// TIA Portal project "Conveyor Speed Control Application with TIA Portal and SCADA" (V16)

(* hardware
DEVICE "PC-System_1"  SIMATIC PC station
   slot 0: "SIMATIC PC station"  Rail  SIMATIC PC-Station  V1.0
      slot 125: "Stationmanager"  Station_Manager  V6.0.4
   slot 1: "HMI_RT_1"  WinCC RT Professional  6AV2 105-0xxxx-xxxx  16.0.0.0
   slot 2: "IE general_1"  IE General  IE_CP  V8.2.0
DEVICE "S7-1200 station_1"  S7-1200 Station
   slot 0: "Rack_0"  S7-1200 Rack  Rack  V1.0
   slot 1: "PLC_1"  CPU 1212C DC/DC/DC  6ES7 212-1AE40-0XB0  V4.4
   slot 2: "AQ 2x14BIT_1"  6ES7 232-4HB30-0XB0  V1.0
   slot 3: "AQ 4x14BIT_1"  SM 1232 AQ4  6ES7 232-4HD30-0XB0  V1.0
DEVICE "HMI_1"  KTP700 Basic PN
   slot 0: "HMI_1"  KTP700 Basic PN  6AV2 123-2GB03-0AX0  16.0.0.0
   slot 1: "HMI_RT_2"  KTP700 Basic PN  6AV2 123-2GB03-0AX0  16.0.0.0
   slot 5: "HMI_1.IE_CP_1"  PROFINET Interface  16.0.0.0
      slot 1: "PROFINET Interface_1"  PROFINET Interface
         slot 1: "Port_1"  Port
*)

// ===== PLC "PLC_1"  CPU 1212C DC/DC/DC =====

VAR_GLOBAL   // PLC tag table "Default tag table"
   "Startup_mem" AT %M10.0 : Bool;
END_VAR

VAR_GLOBAL   // PLC tag table "ANALLOG"
   "BAND2" AT %QW96 : Word;
   "BAND3" AT %QW98 : Int;
   "SİSTEM ÇAŞMA DURUMU" AT %QW30 : Int;
END_VAR

VAR_GLOBAL   // PLC tag table "İnputs"
   "Start_But" AT %I0.0 : Bool;
   "Stop_But" AT %I0.1 : Bool;
   "Start_But_Analog" AT %I0.2 : Bool;
   "Stop_But_Analog" AT %I0.3 : Bool;
   "Start_laması" AT %I0.4 : Bool;
   "Stop_lambası" AT %I0.5 : Bool;
END_VAR

VAR_GLOBAL   // PLC tag table "Outputs"
   "Lamba" AT %Q0.0 : Bool;
   "Band_konveyör" AT %Q0.2 : Bool;
   "Band_konveyör_1" AT %Q0.3 : Bool;
   "Lamba_1" AT %Q0.4 : Bool;
   "konveyör_1" AT %Q0.5 : Bool;
   "konveyör_2" AT %Q0.6 : Bool;
   "konveyör_3" AT %Q0.7 : Bool;
   "konveyör_4" AT %Q1.0 : Bool;
END_VAR

DATA_BLOCK "Datalar"   // DB1
{ S7_Optimized_Access := 'TRUE' }
VERSION : 0.1
   VAR
      Hmi_Start_BUt : Bool;
      Hmi_Stop_BUt : Bool;
      Hmi_jogg_BUt : Bool;
      Band_konveyör : Bool;
      yardımcı_Mem_1 : Bool;
      yardımcı_Mem_2 : Bool;
      Hmi_Toggle_button : Bool;
      Hmi_Azalt_button : Bool;
      Hmi_Artır_button : Bool;
      Hız_değeri : Int;
      band_konveyör_2 : Bool;
      lamba : Bool;
      TEMP_1 : Bool;
      TEMP_2 : Bool;
      TEMP_3 : Bool;
      TEMP_4 : Bool;
      TEMP_5 : Bool;
      KONVEYÖR_HATTI : Struct
         Hmi_Start : Bool;
         Hmi_Stop : Bool;
         Hmi_Merker1 : Bool;
         Sayma_Değeri : Int;
         Hmi_Start_Analog : Bool;
         Hmi_Stop_Analog : Bool;
         Start_Stop_button : Bool;
         Start_Stop_Mem : Bool;
         "Sistem_durum bilgisi" : Int;
      END_STRUCT;
   END_VAR
BEGIN
END_DATA_BLOCK

// folder: System blocks/Program resources

DATA_BLOCK "time_1"   // DB2
{ S7_Optimized_Access := 'TRUE' }
AUTHOR : Simatic
FAMILY : IEC
NAME : IEC_TMR
VERSION : 1.0
// stored: InstanceOfName IEC_TIMER
"IEC_TIMER"
BEGIN
END_DATA_BLOCK

DATA_BLOCK "time_2"   // DB3
{ S7_Optimized_Access := 'TRUE' }
AUTHOR : Simatic
FAMILY : IEC
NAME : IEC_TMR
VERSION : 1.0
// stored: InstanceOfName IEC_TIMER
"IEC_TIMER"
BEGIN
END_DATA_BLOCK

// folder: (top level)

FUNCTION "üretim Hattı 2" : Void   // FC1, LAD
{ S7_Optimized_Access := 'TRUE' }
VERSION : 0.1
BEGIN

REGION Network 1
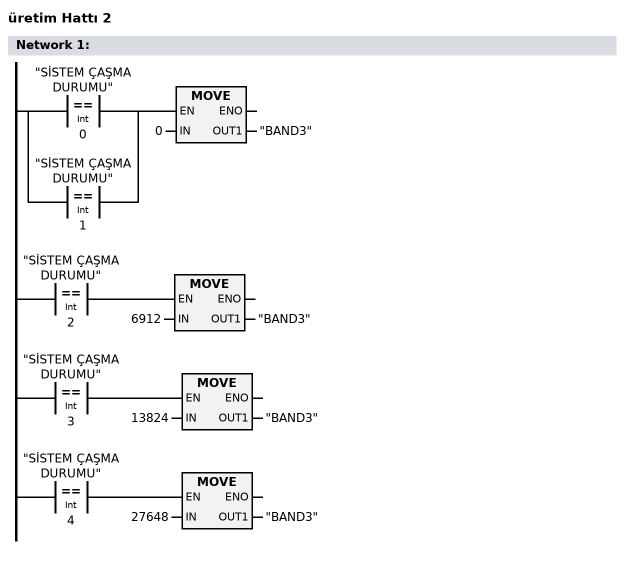
   RUNG wire#powerrail
      { S7_Templates := "SrcType := Int" } EQ_Contact(in1 := "SİSTEM ÇAŞMA DURUMU", in2 := 0)
      wire#w1
      Move(in := 0, out1 => "BAND3")
   END_RUNG
   RUNG wire#powerrail
      { S7_Templates := "SrcType := Int" } EQ_Contact(in1 := "SİSTEM ÇAŞMA DURUMU", in2 := 1)
   END_RUNG wire#w1
   RUNG wire#powerrail
      { S7_Templates := "SrcType := Int" } EQ_Contact(in1 := "SİSTEM ÇAŞMA DURUMU", in2 := 2)
      Move(in := 6912, out1 => "BAND3")
   END_RUNG
   RUNG wire#powerrail
      { S7_Templates := "SrcType := Int" } EQ_Contact(in1 := "SİSTEM ÇAŞMA DURUMU", in2 := 3)
      Move(in := 13824, out1 => "BAND3")
   END_RUNG
   RUNG wire#powerrail
      { S7_Templates := "SrcType := Int" } EQ_Contact(in1 := "SİSTEM ÇAŞMA DURUMU", in2 := 4)
      Move(in := 27648, out1 => "BAND3")
   END_RUNG
   // the same network as SCL:
   IF ("SİSTEM ÇAŞMA DURUMU" = 0) OR ("SİSTEM ÇAŞMA DURUMU" = 1) THEN "BAND3" := 0; END_IF;
   IF "SİSTEM ÇAŞMA DURUMU" = 2 THEN "BAND3" := 6912; END_IF;
   IF "SİSTEM ÇAŞMA DURUMU" = 3 THEN "BAND3" := 13824; END_IF;
   IF "SİSTEM ÇAŞMA DURUMU" = 4 THEN "BAND3" := 27648; END_IF;
END_REGION
END_FUNCTION

FUNCTION "Üretin_hattı_3" : Void   // FC2, LAD
{ S7_Optimized_Access := 'TRUE' }
VERSION : 0.1
BEGIN

REGION Network 1: Sistem Start Stop
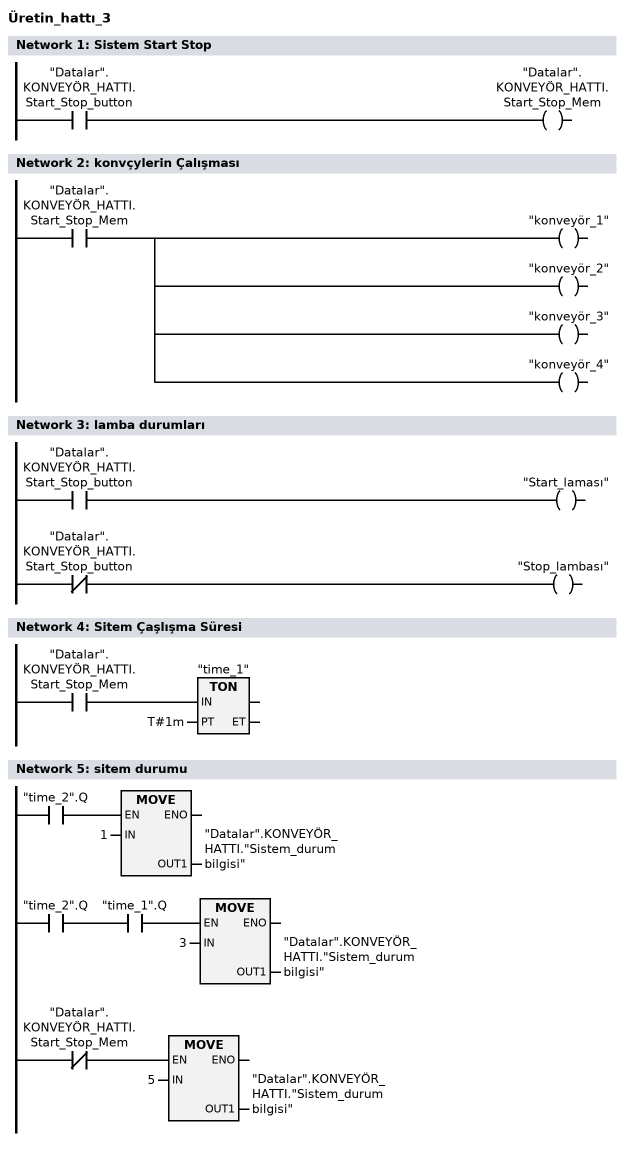
   RUNG wire#powerrail
      Contact( "Datalar".KONVEYÖR_HATTI.Start_Stop_button )
      Coil( "Datalar".KONVEYÖR_HATTI.Start_Stop_Mem )
   END_RUNG
   // the same network as SCL:
   "Datalar".KONVEYÖR_HATTI.Start_Stop_Mem := "Datalar".KONVEYÖR_HATTI.Start_Stop_button;
END_REGION

REGION Network 2: konvçylerin Çalışması
   RUNG wire#powerrail
      Contact( "Datalar".KONVEYÖR_HATTI.Start_Stop_Mem )
      wire#w1
      Coil( "konveyör_1" )
   END_RUNG
   RUNG wire#w1
      Coil( "konveyör_2" )
   END_RUNG
   RUNG wire#w1
      Coil( "konveyör_3" )
   END_RUNG
   RUNG wire#w1
      Coil( "konveyör_4" )
   END_RUNG
   // the same network as SCL:
   "konveyör_1" := "Datalar".KONVEYÖR_HATTI.Start_Stop_Mem;
   "konveyör_2" := "Datalar".KONVEYÖR_HATTI.Start_Stop_Mem;
   "konveyör_3" := "Datalar".KONVEYÖR_HATTI.Start_Stop_Mem;
   "konveyör_4" := "Datalar".KONVEYÖR_HATTI.Start_Stop_Mem;
END_REGION

REGION Network 3: lamba durumları
   RUNG wire#powerrail
      Contact( "Datalar".KONVEYÖR_HATTI.Start_Stop_button )
      Coil( "Start_laması" )
   END_RUNG
   RUNG wire#powerrail
      I_Contact( "Datalar".KONVEYÖR_HATTI.Start_Stop_button )
      Coil( "Stop_lambası" )
   END_RUNG
   // the same network as SCL:
   "Start_laması" := "Datalar".KONVEYÖR_HATTI.Start_Stop_button;
   "Stop_lambası" := NOT "Datalar".KONVEYÖR_HATTI.Start_Stop_button;
END_REGION

REGION Network 4: Sitem Çaşlışma Süresi
   "time_1".TON(IN := "Datalar".KONVEYÖR_HATTI.Start_Stop_Mem, PT := T#1m);
END_REGION

REGION Network 5: sitem durumu
   RUNG wire#powerrail
      Contact( "time_2".Q )
      Move(in := 1, out1 => "Datalar".KONVEYÖR_HATTI."Sistem_durum bilgisi")
   END_RUNG
   RUNG wire#powerrail
      Contact( "time_2".Q )
      Contact( "time_1".Q )
      Move(in := 3, out1 => "Datalar".KONVEYÖR_HATTI."Sistem_durum bilgisi")
   END_RUNG
   RUNG wire#powerrail
      I_Contact( "Datalar".KONVEYÖR_HATTI.Start_Stop_Mem )
      Move(in := 5, out1 => "Datalar".KONVEYÖR_HATTI."Sistem_durum bilgisi")
   END_RUNG
   // the same network as SCL:
   IF "time_2".Q THEN "Datalar".KONVEYÖR_HATTI."Sistem_durum bilgisi" := 1; END_IF;
   IF "time_2".Q AND "time_1".Q THEN "Datalar".KONVEYÖR_HATTI."Sistem_durum bilgisi" := 3; END_IF;
   IF NOT "Datalar".KONVEYÖR_HATTI.Start_Stop_Mem THEN
       "Datalar".KONVEYÖR_HATTI."Sistem_durum bilgisi" := 5;
   END_IF;
END_REGION
END_FUNCTION

ORGANIZATION_BLOCK "Main"   // OB1, LAD, ProgramCycle
TITLE = "Main Program Sweep (Cycle)"
{ S7_Optimized_Access := 'TRUE' }
VERSION : 0.1
   VAR_INPUT
      Initial_Call : Bool;   // Initial call of this OB
      Remanence : Bool;   // =True, if remanent data are available
   END_VAR
   VAR_TEMP   // added for the SCL form of the ladder/FBD networks
      _w1 : Bool;
      _w2 : Bool;
   END_VAR
BEGIN

REGION Network 1: ÜRETİM HATTI 2
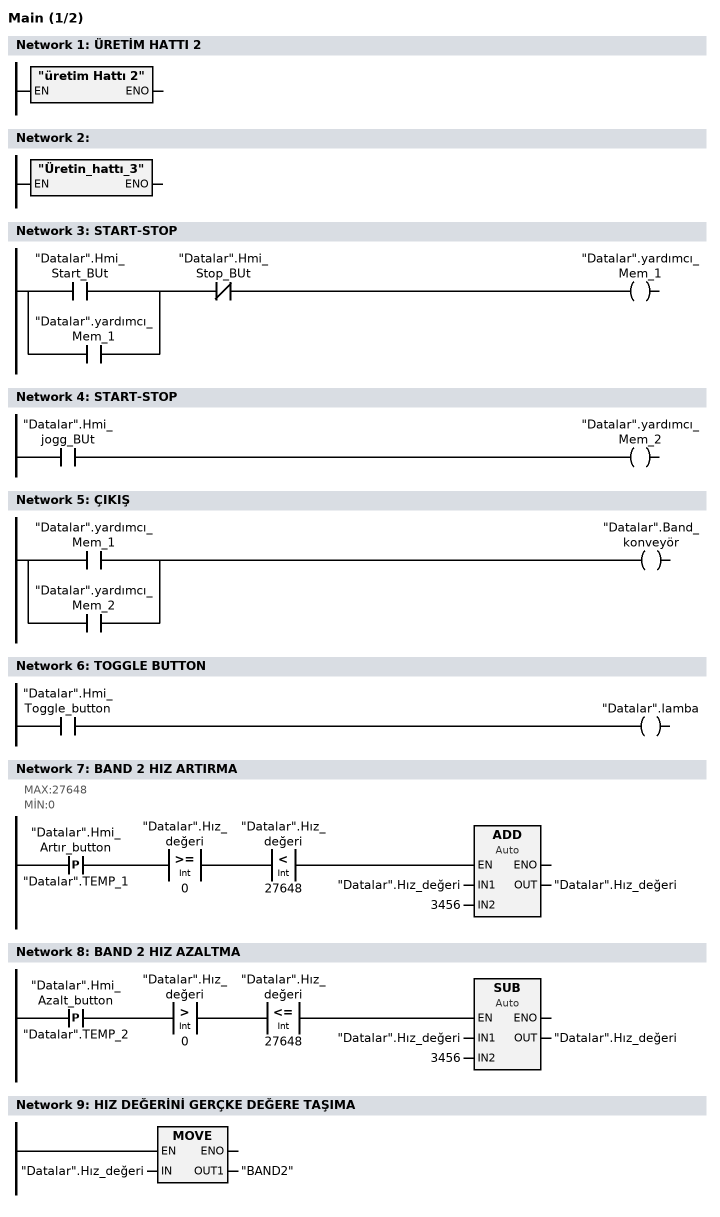
   RUNG wire#powerrail
      "üretim Hattı 2"()
   END_RUNG
   // the same network as SCL:
   "üretim Hattı 2"();
END_REGION

REGION Network 2
   RUNG wire#powerrail
      "Üretin_hattı_3"()
   END_RUNG
   // the same network as SCL:
   "Üretin_hattı_3"();
END_REGION

REGION Network 3: START-STOP
   RUNG wire#powerrail
      Contact( "Datalar".Hmi_Start_BUt )
      wire#w1
      I_Contact( "Datalar".Hmi_Stop_BUt )
      Coil( "Datalar".yardımcı_Mem_1 )
   END_RUNG
   RUNG wire#powerrail
      Contact( "Datalar".yardımcı_Mem_1 )
   END_RUNG wire#w1
   // the same network as SCL:
   "Datalar".yardımcı_Mem_1 := ("Datalar".Hmi_Start_BUt OR "Datalar".yardımcı_Mem_1) AND NOT "Datalar".Hmi_Stop_BUt;
END_REGION

REGION Network 4: START-STOP
   RUNG wire#powerrail
      Contact( "Datalar".Hmi_jogg_BUt )
      Coil( "Datalar".yardımcı_Mem_2 )
   END_RUNG
   // the same network as SCL:
   "Datalar".yardımcı_Mem_2 := "Datalar".Hmi_jogg_BUt;
END_REGION

REGION Network 5: ÇIKIŞ
   RUNG wire#powerrail
      Contact( "Datalar".yardımcı_Mem_1 )
      wire#w1
      Coil( "Datalar".Band_konveyör )
   END_RUNG
   RUNG wire#powerrail
      Contact( "Datalar".yardımcı_Mem_2 )
   END_RUNG wire#w1
   // the same network as SCL:
   "Datalar".Band_konveyör := "Datalar".yardımcı_Mem_1 OR "Datalar".yardımcı_Mem_2;
END_REGION

REGION Network 6: TOGGLE BUTTON
   RUNG wire#powerrail
      Contact( "Datalar".Hmi_Toggle_button )
      Coil( "Datalar".lamba )
   END_RUNG
   // the same network as SCL:
   "Datalar".lamba := "Datalar".Hmi_Toggle_button;
END_REGION

REGION Network 7: BAND 2 HIZ ARTIRMA
   // MAX:27648
   // MİN:0
   RUNG wire#powerrail
      P_Contact(operand := "Datalar".Hmi_Artır_button, bit := "Datalar".TEMP_1)
      { S7_Templates := "SrcType := Int" } GE_Contact(in1 := "Datalar".Hız_değeri, in2 := 0)
      { S7_Templates := "SrcType := Int" } LT_Contact(in1 := "Datalar".Hız_değeri, in2 := 27648)
      Add(in1 := "Datalar".Hız_değeri, in2 := 3456, out => "Datalar".Hız_değeri)
   END_RUNG
   // the same network as SCL:
   #_w1 := "Datalar".Hmi_Artır_button AND NOT "Datalar".TEMP_1;   // rising edge of "Datalar".Hmi_Artır_button
   "Datalar".TEMP_1 := "Datalar".Hmi_Artır_button;
   IF #_w1 AND ("Datalar".Hız_değeri >= 0) AND ("Datalar".Hız_değeri < 27648) THEN
       "Datalar".Hız_değeri := "Datalar".Hız_değeri + 3456;
   END_IF;
END_REGION

REGION Network 8: BAND 2 HIZ AZALTMA
   RUNG wire#powerrail
      P_Contact(operand := "Datalar".Hmi_Azalt_button, bit := "Datalar".TEMP_2)
      { S7_Templates := "SrcType := Int" } GT_Contact(in1 := "Datalar".Hız_değeri, in2 := 0)
      { S7_Templates := "SrcType := Int" } LE_Contact(in1 := "Datalar".Hız_değeri, in2 := 27648)
      Sub(in1 := "Datalar".Hız_değeri, in2 := 3456, out => "Datalar".Hız_değeri)
   END_RUNG
   // the same network as SCL:
   #_w1 := "Datalar".Hmi_Azalt_button AND NOT "Datalar".TEMP_2;   // rising edge of "Datalar".Hmi_Azalt_button
   "Datalar".TEMP_2 := "Datalar".Hmi_Azalt_button;
   IF #_w1 AND ("Datalar".Hız_değeri > 0) AND ("Datalar".Hız_değeri <= 27648) THEN
       "Datalar".Hız_değeri := "Datalar".Hız_değeri - 3456;
   END_IF;
END_REGION

REGION Network 9: HIZ DEĞERİNİ GERÇKE DEĞERE TAŞIMA
   RUNG wire#powerrail
      Move(in := "Datalar".Hız_değeri, out1 => "BAND2")
   END_RUNG
   // the same network as SCL:
   "BAND2" := "Datalar".Hız_değeri;
END_REGION

REGION Network 10: KONYEYÖR HATTINI ÇALIŞTIRMA 1
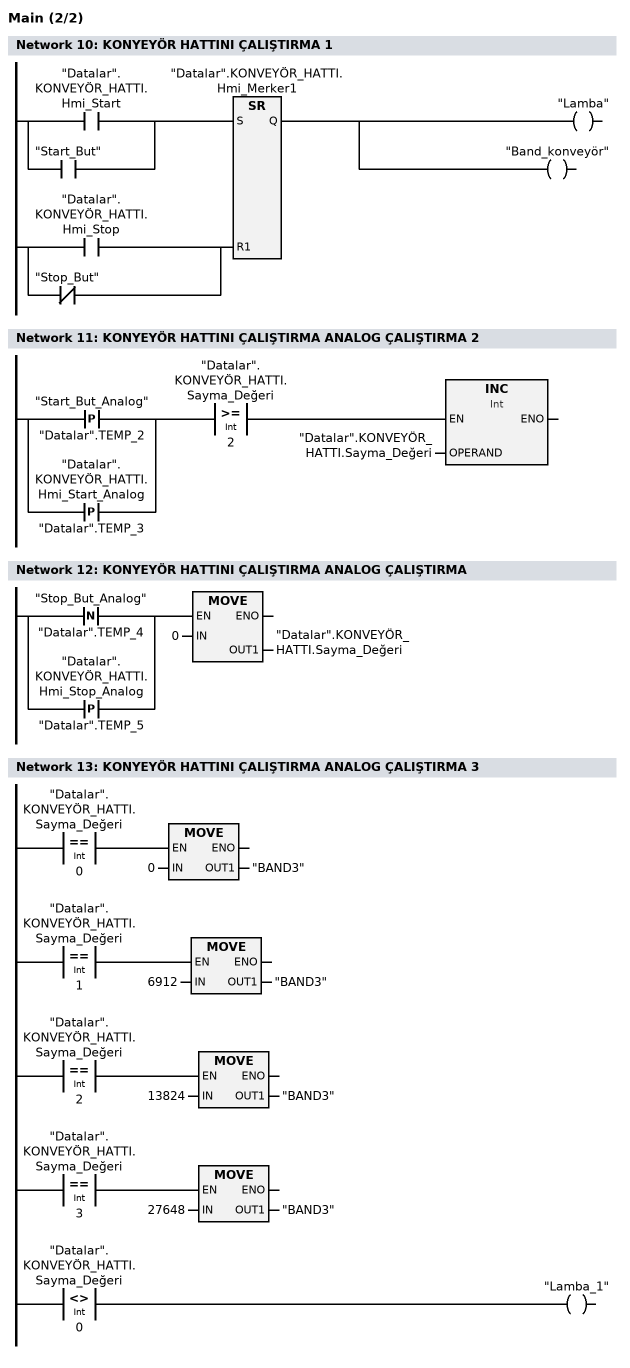
   RUNG wire#powerrail
      Contact( "Datalar".KONVEYÖR_HATTI.Hmi_Start )
      wire#w1
      S_SR(operand := "Datalar".KONVEYÖR_HATTI.Hmi_Merker1, r1 := wire#w2)
      wire#w3
      Coil( "Lamba" )
   END_RUNG
   RUNG wire#powerrail
      Contact( "Start_But" )
   END_RUNG wire#w1
   RUNG wire#powerrail
      Contact( "Datalar".KONVEYÖR_HATTI.Hmi_Stop )
   END_RUNG wire#w2
   RUNG wire#powerrail
      I_Contact( "Stop_But" )
   END_RUNG wire#w2
   RUNG wire#w3
      Coil( "Band_konveyör" )
   END_RUNG
   // the same network as SCL:
   IF "Datalar".KONVEYÖR_HATTI.Hmi_Start OR "Start_But" THEN
       "Datalar".KONVEYÖR_HATTI.Hmi_Merker1 := TRUE;   // SR flip-flop
   END_IF;
   IF "Datalar".KONVEYÖR_HATTI.Hmi_Stop OR NOT "Stop_But" THEN
       "Datalar".KONVEYÖR_HATTI.Hmi_Merker1 := FALSE;
   END_IF;
   "Lamba" := "Datalar".KONVEYÖR_HATTI.Hmi_Merker1;
   "Band_konveyör" := "Datalar".KONVEYÖR_HATTI.Hmi_Merker1;
END_REGION

REGION Network 11: KONYEYÖR HATTINI ÇALIŞTIRMA ANALOG ÇALIŞTIRMA 2
   RUNG wire#powerrail
      P_Contact(operand := "Start_But_Analog", bit := "Datalar".TEMP_2)
      wire#w1
      { S7_Templates := "SrcType := Int" } GE_Contact(in1 := "Datalar".KONVEYÖR_HATTI.Sayma_Değeri, in2 := 2)
      { S7_Templates := "DestType := Int" } Inc( "Datalar".KONVEYÖR_HATTI.Sayma_Değeri )
   END_RUNG
   RUNG wire#powerrail
      P_Contact(operand := "Datalar".KONVEYÖR_HATTI.Hmi_Start_Analog, bit := "Datalar".TEMP_3)
   END_RUNG wire#w1
   // the same network as SCL:
   #_w1 := "Start_But_Analog" AND NOT "Datalar".TEMP_2;   // rising edge of "Start_But_Analog"
   "Datalar".TEMP_2 := "Start_But_Analog";
   #_w2 := "Datalar".KONVEYÖR_HATTI.Hmi_Start_Analog AND NOT "Datalar".TEMP_3;   // rising edge of "Datalar".KONVEYÖR_HATTI.Hmi_Start_Analog
   "Datalar".TEMP_3 := "Datalar".KONVEYÖR_HATTI.Hmi_Start_Analog;
   IF (#_w1 OR #_w2) AND ("Datalar".KONVEYÖR_HATTI.Sayma_Değeri >= 2) THEN
       "Datalar".KONVEYÖR_HATTI.Sayma_Değeri := "Datalar".KONVEYÖR_HATTI.Sayma_Değeri + 1;
   END_IF;
END_REGION

REGION Network 12: KONYEYÖR HATTINI ÇALIŞTIRMA ANALOG ÇALIŞTIRMA
   RUNG wire#powerrail
      N_Contact(operand := "Stop_But_Analog", bit := "Datalar".TEMP_4)
      wire#w1
      Move(in := 0, out1 => "Datalar".KONVEYÖR_HATTI.Sayma_Değeri)
   END_RUNG
   RUNG wire#powerrail
      P_Contact(operand := "Datalar".KONVEYÖR_HATTI.Hmi_Stop_Analog, bit := "Datalar".TEMP_5)
   END_RUNG wire#w1
   // the same network as SCL:
   #_w1 := NOT "Stop_But_Analog" AND "Datalar".TEMP_4;   // falling edge of "Stop_But_Analog"
   "Datalar".TEMP_4 := "Stop_But_Analog";
   #_w2 := "Datalar".KONVEYÖR_HATTI.Hmi_Stop_Analog AND NOT "Datalar".TEMP_5;   // rising edge of "Datalar".KONVEYÖR_HATTI.Hmi_Stop_Analog
   "Datalar".TEMP_5 := "Datalar".KONVEYÖR_HATTI.Hmi_Stop_Analog;
   IF #_w1 OR #_w2 THEN "Datalar".KONVEYÖR_HATTI.Sayma_Değeri := 0; END_IF;
END_REGION

REGION Network 13: KONYEYÖR HATTINI ÇALIŞTIRMA ANALOG ÇALIŞTIRMA 3
   RUNG wire#powerrail
      { S7_Templates := "SrcType := Int" } EQ_Contact(in1 := "Datalar".KONVEYÖR_HATTI.Sayma_Değeri, in2 := 0)
      Move(in := 0, out1 => "BAND3")
   END_RUNG
   RUNG wire#powerrail
      { S7_Templates := "SrcType := Int" } EQ_Contact(in1 := "Datalar".KONVEYÖR_HATTI.Sayma_Değeri, in2 := 1)
      Move(in := 6912, out1 => "BAND3")
   END_RUNG
   RUNG wire#powerrail
      { S7_Templates := "SrcType := Int" } EQ_Contact(in1 := "Datalar".KONVEYÖR_HATTI.Sayma_Değeri, in2 := 2)
      Move(in := 13824, out1 => "BAND3")
   END_RUNG
   RUNG wire#powerrail
      { S7_Templates := "SrcType := Int" } EQ_Contact(in1 := "Datalar".KONVEYÖR_HATTI.Sayma_Değeri, in2 := 3)
      Move(in := 27648, out1 => "BAND3")
   END_RUNG
   RUNG wire#powerrail
      { S7_Templates := "SrcType := Int" } NE_Contact(in1 := "Datalar".KONVEYÖR_HATTI.Sayma_Değeri, in2 := 0)
      Coil( "Lamba_1" )
   END_RUNG
   // the same network as SCL:
   IF "Datalar".KONVEYÖR_HATTI.Sayma_Değeri = 0 THEN "BAND3" := 0; END_IF;
   IF "Datalar".KONVEYÖR_HATTI.Sayma_Değeri = 1 THEN "BAND3" := 6912; END_IF;
   IF "Datalar".KONVEYÖR_HATTI.Sayma_Değeri = 2 THEN "BAND3" := 13824; END_IF;
   IF "Datalar".KONVEYÖR_HATTI.Sayma_Değeri = 3 THEN "BAND3" := 27648; END_IF;
   "Lamba_1" := "Datalar".KONVEYÖR_HATTI.Sayma_Değeri <> 0;
END_REGION
END_ORGANIZATION_BLOCK

ORGANIZATION_BLOCK "Startup"   // OB100, LAD, Startup
TITLE = "Complete Restart"
{ S7_Optimized_Access := 'TRUE' }
VERSION : 0.1
   VAR_INPUT
      LostRetentive : Bool;   // True if retentive data are lost
      LostRTC : Bool;   // True if date and time are lost
   END_VAR
BEGIN

REGION Network 1
   // plc Stop modula alıp terkara run veririsek 25saniye sonra run oluca
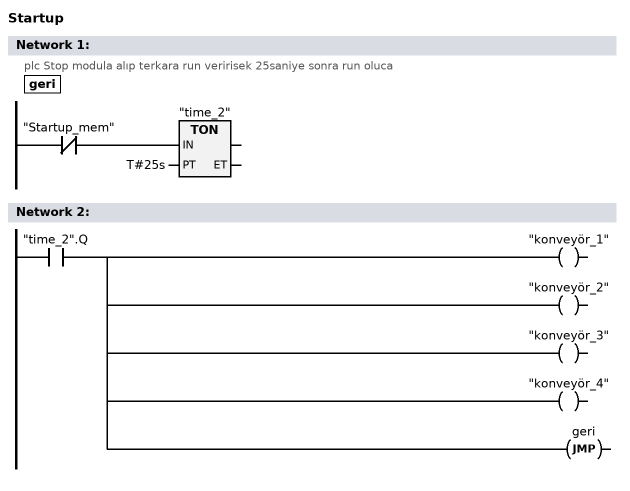
   geri:
   "time_2".TON(IN := NOT "Startup_mem", PT := T#25s);
END_REGION

REGION Network 2
   RUNG wire#powerrail
      Contact( "time_2".Q )
      wire#w1
      Coil( "konveyör_1" )
   END_RUNG
   RUNG wire#w1
      Coil( "konveyör_2" )
   END_RUNG
   RUNG wire#w1
      Coil( "konveyör_3" )
   END_RUNG
   RUNG wire#w1
      Coil( "konveyör_4" )
   END_RUNG
   RUNG wire#w1
      JumpCoil( geri )
   END_RUNG
   // the same network as SCL:
   "konveyör_1" := "time_2".Q;
   "konveyör_2" := "time_2".Q;
   "konveyör_3" := "time_2".Q;
   "konveyör_4" := "time_2".Q;
   IF "time_2".Q THEN GOTO geri; END_IF;
END_REGION
END_ORGANIZATION_BLOCK

(* ===== HMI "HMI_RT_1" =====
system functions are stored by id; their names below are inferred from use
connection "HMI_Connection_1": S71200_TCP_IP, SCADA_S7_1200

HMI tags "Default tag table"
   "a" : Bool = PLC a AT %I0.0, 500 ms
   "Datalar_Hmi_Start_BUt" : Bool = PLC Datalar.Hmi_Start_BUt, 500 ms
   "Datalar_Hmi_Stop_BUt" : Bool = PLC Datalar.Hmi_Stop_BUt, 500 ms
   "Datalar_Hmi_jogg_BUt" : Bool = PLC Datalar.Hmi_jogg_BUt, 500 ms
   "Datalar_Hmi_Toggle_button" : Bool = PLC Datalar.Hmi_Toggle_button, 500 ms
   "Datalar_Hmi_Artır_button" : Bool = PLC Datalar.Hmi_Artır_button, 500 ms
   "Datalar_Hmi_Azalt_button" : Bool = PLC Datalar.Hmi_Azalt_button, 500 ms
   "Datalar_KONVEYÖR_HATTI_Hmi_Start" : Bool = PLC Datalar.KONVEYÖR_HATTI.Hmi_Start, 500 ms
   "Datalar_KONVEYÖR_HATTI_Hmi_Stop" : Bool = PLC Datalar.KONVEYÖR_HATTI.Hmi_Stop, 500 ms
   "Lamba" : Bool = PLC Lamba AT %Q0.0, 500 ms
   "Band_konveyör" : Bool = PLC Band_konveyör AT %Q0.2, 500 ms
   "BAND3" : Int = PLC BAND3 AT %QW98, 500 ms
   "SİSTEMÇAŞMADURUMU" : Int = PLC "SİSTEM ÇAŞMA DURUMU" AT %QW30, 500 ms
   "Datalar_KONVEYÖR_HATTI_Sistem_durumbilgisi" : Int = PLC Datalar.KONVEYÖR_HATTI."Sistem_durum bilgisi", 500 ms
   "Datalar_KONVEYÖR_HATTI_Start_Stop_button" : Bool = PLC Datalar.KONVEYÖR_HATTI.Start_Stop_button, 500 ms

screen "Ana Sayfa" 1024x768
   Button "Button_1" at 118,107 size 107x63; TextOff 'START BUT'
   Button "Button_2" at 250,109 size 107x63; TextOff 'STOP BUT'
      on PressLeft: SetBit("Datalar_Hmi_Stop_BUt")
      on ReleaseLeft: ResetBit("Datalar_Hmi_Stop_BUt")
   Button "Button_3" at 390,109 size 107x63; TextOff 'JOGG BUT'
      on PressLeft: SetBit("Datalar_Hmi_jogg_BUt")
      on ReleaseLeft: ResetBit("Datalar_Hmi_jogg_BUt")
   RoundButton "Round button_1" at 299,306 size 93x93; Text 'TOGGLE BUTTON'
      on Click: InvertBit("Datalar_Hmi_Toggle_button")
   TextField "Text field_1" at 262,17 size 144x23; Text 'BUTTON TİPLERİ'
   Button "Button_4" at 156,282 size 76x60; TextOff 'Text'; PictureOff "Up_Arrow"
      on PressLeft: SetBit("Datalar_Hmi_Artır_button")
      on ReleaseLeft: ResetBit("Datalar_Hmi_Artır_button")
   Button "Button_5" at 162,399 size 72x66; TextOff 'Text'; PictureOff "Down_Arrow"
      on PressLeft: SetBit("Datalar_Hmi_Azalt_button")
      on ReleaseLeft: ResetBit("Datalar_Hmi_Azalt_button")
   TextField "Text field_2" at 159,246 size 80x21; Text 'HIZ ARTIR'
   TextField "Text field_3" at 159,369 size 82x21; Text 'HIZ AZALT'

screen "Üretim Hattı" 1024x768
   GraphicView "Graphic view_1" at 155,46 size 299x183; Picture "Graphic_1"
   TextField "Text field_1" at 259,15 size 102x19; Text 'Üretim Hattı'
   Button "Button_1" at 512,70 size 99x52; TextOff 'Start'
      on PressLeft: SetBit("Datalar_KONVEYÖR_HATTI_Hmi_Start")
      on ReleaseLeft: ResetBit("Datalar_KONVEYÖR_HATTI_Hmi_Start")
   Button "Button_2" at 686,70 size 99x52; TextOff 'Stop'
      on PressLeft: SetBit("Datalar_KONVEYÖR_HATTI_Hmi_Stop")
      on ReleaseLeft: ResetBit("Datalar_KONVEYÖR_HATTI_Hmi_Stop")
   GraphicView "Graphic view_2" at 258,112 size 97x127; Picture "Graphic_2"
   Circle "Circle_1" at 268,132 size 25x25
      Visibility <- "Lamba"
      Appearance <- "BAND3"
   Circle "Circle_2" at 310,132 size 24x24
      Appearance <- "BAND3"
   TextField "Text field_2" at 259,241 size 110x19; Text 'sistem Çalışıyor'
      Visibility <- "Band_konveyör"
   TextField "Text field_3" at 259,271 size 108x19; Text 'sistem Duruyor'
      Visibility <- "Band_konveyör"
   ListBox "List box_1" at 422,171 size 300x15; Text0 'Text1'
      SelectedIndex <- "BAND3"
      PropertyAnimation0 <- "BAND3"

screen "Üreti Hattı_2" 1024x768
   GraphicView "Graphic view_1" at 155,46 size 299x183; Picture "Graphic_1"
   TextField "Text field_1" at 259,15 size 102x19; Text 'Üretim Hattı'
   GraphicView "Graphic view_2" at 258,112 size 97x127; Picture "Graphic_2"
   Circle "Circle_1" at 268,132 size 25x25
      Visibility <- "Lamba"
      Appearance <- "BAND3"
   Circle "Circle_2" at 310,132 size 24x24
      Appearance <- "BAND3"
   ListBox "List box_1" at 109,241 size 461x68; Text0 'SİSTEM DURUYOR'; Text1 'SİSTEM YAVAŞ HIZDA ÇALIŞIYOR'; Text2 'SİSTEM ORTA HIZDA ÇALIŞIYOR'; Text3 'SİSTEM YÜKSEK HIZDA ÇALIŞIYOR'
      SelectedIndex <- "SİSTEMÇAŞMADURUMU"
   Button "Button_1" at 509,60 size 124x65; TextOff 'Start'
   Button "Button_2" at 672,57 size 124x65; TextOff 'Stop'
   ComboBox "Combo box_1" at 120,339 size 439x30; Text0 'SİSTEM DURUYOR'; Text1 'SİSTEM YAVAŞ HIZDA ÇALIŞIYOR'; Text2 'SİSTEM ORTA HIZDA ÇALIŞIYOR'; Text3 'SİSTEM YÜKSEK HIZDA ÇALIŞIYOR'
      SelectedIndex <- "SİSTEMÇAŞMADURUMU"

screen "Üretim hattı_3" 1024x768
   RoundButton "Round button_1" at 42,117 size 83x83; Text 'Start Stop'
      on Click: InvertBit("Datalar_KONVEYÖR_HATTI_Start_Stop_button")
   GraphicView "Graphic view_1" at 200,35 size 299x183; Picture "Graphic_1"
   GraphicView "Graphic view_2" at 303,101 size 97x127; Picture "Graphic_2"
   CheckBox "Check box_1" at 94,266 size 236x93; Text0 'Sistem ilk konuma Alındı'; Text1 'Sistem Bir dk dan fazla çalıştı'; Text2 'Sistem Durdu'
      ProcessValue <- "Datalar_KONVEYÖR_HATTI_Sistem_durumbilgisi"
   TextField "Text field_1" at 111,243 size 90x19; Text 'Onay Kutusu'
*)

(* ===== HMI "HMI_RT_2" =====
system functions are stored by id; their names below are inferred from use
connection "HMI_Connection_2": ETHERNET, SMART_S7_1200_OMS

HMI tags "Default tag table"
   "Tag_ScreenNumber" : UInt, internal

Template "Template_1" 800x480
   Button "Exit" at 714,429 size 71x50; TextOff 'Exit'; PictureOff "ExitRuntime_KTP700_Basic_PN_TR"; PictureOn "ExitRuntime_KTP700_Basic_PN_TR"
      on Release: StopRuntime(0)
   Button "Template_Button" at 614,429 size 71x50; TextOff 'Text'
   Button "Template_Button_1" at 514,429 size 71x50; TextOff 'Text'
   Button "Template_Button_2" at 414,429 size 71x50; TextOff 'Text'
   Button "Template_Button_3" at 314,429 size 71x50; TextOff 'Text'
   Button "Template_Button_4" at 214,429 size 71x50; TextOff 'Text'
   Button "Template_Button_5" at 114,429 size 71x50; TextOff 'Text'
   Button "Start screen" at 14,429 size 71x50; TextOff 'Start screen'; PictureOff "NavigateHome_KTP700_Basic_PN_TR"; PictureOn "NavigateHome_KTP700_Basic_PN_TR"
      on Release: ActivateScreen("Root screen", 0)
   SymbolicIOField "Symbolic_IO_Field_Screen" at 93,9 size 600x33; TextOff '0'; TextOn '1'; TextList "TextList_ScreenNames"
      ProcessValue <- "Tag_ScreenNumber"
      on Change: ActivateScreenByNumber("Tag_ScreenNumber", 0)
   DateTimeField "HmiScreenItemData" at 695,25 size 105x25
   DateTimeField "HmiScreenItemData_1" at 695,0 size 105x25
   GraphicView "Logo" at 0,0 size 91x51; Picture "Logo of HMI_1"

screen "Root screen" 800x480, template "Template_1"
   on GenerateScreen: SetTag("Tag_ScreenNumber", 1)
*)